(* PLC project A2ServodriveLibrary, Delta Electronics, Inc. DIADesigner-AX DIADesigner-AX 1.3, author Piotr Gliszczyński *)
(* stored: creationDateTime 2022-11-07T17:46:50.8449516, version 3.5.15.30, modificationDateTime 2022-11-07T17:45:55.5007525, organization Induprogress sp. z o.o *)
(* Library for using A2 via CiA402. For now enum for error codes processing is available. *)

{attribute 'qualified_only'}
{attribute 'strict'}
{attribute 'to_string'}
TYPE DriveA2Error : (NO_ERROR := 0, OVER_CURRENT_AL001 := 16#1, OVER_VOLTAGE_AL002 := 16#2, UNDER_VOLTAGE_AL003 := 16#3, MOTOR_COMBINATION_ERROR_AL004 := 16#4, REGENERATION_ERROR_AL005 := 16#5, OVERLOAD_AL006 := 16#6, OVERSPEED_AL007 := 16#7, ABNORMAL_PULSE_COMMAND_AL008 := 16#8, EXCESSIVE_DEVIATION_OF_POSITION_COMMAND_AL009 := 16#9, ENCODER_ERROR_AL011 := 16#11, ADJUSTMENT_ERROR_AL012 := 16#12, EMERGENCY_STOP_AL013 := 16#13, REVERSE_LIMIT_ERROR_AL014 := 16#14, FORWARD_LIMIT_ERROR_AL015 := 16#15, IGBT_OVERHEAT_AL016 := 16#16, ABNORMAL_ERROR_AL017 := 16#17, ABNORMAL_SIGNAL_OUTPUT_AL018 := 16#18, SERIAL_COMMUNICATION_ERROR_AL019 := 16#19, SERIAL_COMMUNICATION_TIME_OUT_AL020 := 16#20, MAIN_CIRCUIT_POWER_LACK_PHASE_AL022 := 16#22, EARLY_WARNING_FOR_OVERLOAD_AL023 := 16#23, ENCODER_INITIAL_MAGNETIC_FIELD_ERROR_AL024 := 16#24, THE_INTERNAL_OF_THE_ENCODER_IS_IN_ERROR_AL025 := 16#25, UNRELIABLE_INTERNAL_DATA_OF_THE_ENCODER_AL026 := 16#26, THE_INTERNAL_OF_THE_IS_IN_ERROR_AL027 := 16#27, ENCODER_VOLTAGE_ERROR_AL028 := 16#28, GRAY_CODE_ERROR_AL029 := 16#29, MOTOR_CRASH_ERROR_AL030 := 16#30, INCORRECT_WIRING_OF_THE_MOTOR_POWER_LINE_UVW_GND_AL031 := 16#31, INTERNAL_COMMUNICATION_OF_THE_ENCODER_IS_IN_ERROR_AL034 := 16#34, ENCODER_TEMPERATURE_EXCEEDS_THE_PROTECTIVE_RANGE_AL035 := 16#35, EXCESSIVE_DEVIATION_OF_FULL_CLOSED_LOOP_AL040 := 16#40, COMMUNICATION_OF_LINEAR_SCALE_IS_BREAKDOWN_AL041 := 16#41, ANALOG_INPUT_VOLTAGE_ERROR_AL042 := 16#42, WARNING_OF_SERVODRIVE_FUNCTION_OVERLOAD_AL043 := 16#43, WRONG_SETTING_OF_E_GEAR_RATIO_AL045 := 16#45, THE_ABSOLUTE_POSITION_IS_LOST_AL060 := 16#60, ENCODER_UNDER_VOLTAGE_AL061 := 16#61, THE_MULTITURN_OF_ABSOLUTE_ENCODER_OVERFLOWS_AL062 := 16#62, ENCODER_TEMPERATURE_WARNING_AL067 := 16#67, ABSOLUTE_DATA_TRANSMITTED_VIA_IO_IS_IN_ERROR_AL068 := 16#68, WRONG_MOTOR_TYPE_AL069 := 16#69, THE_ABSOLUTE_COORDINATE_HAS_NOT_BEEN_INITIALIZED_AL06A := 16#6A, ENCODER_DOES_NOT_COMPLETE_THE_COMMAND_AL070 := 16#70, ENCODER_OVERSPEED_AL072 := 16#72, ENCODER_MEMORY_ERROR_AL073 := 16#73, ABSOLUTE_ENCODER_SINGLE_TURN_POSITION_ERROR_AL074 := 16#74, ABSOLUTE_ENCODER_POSITION_ERROR_AL075 := 16#75, ENCODER_COMPUTING_ERROR_AL077 := 16#77, ENCODER_PARAMETER_ERROR_AL079 := 16#79, LOSS_OF_ENCODER_Z_PULSE_AL07A := 16#7A, ENCODER_MEMORY_BUSY_AL07B := 16#7B, COMMAND_TO_CLEAR_THE_ABSOLUTE_POSITION_ISSUED_WHEN_MOTOR_SPEED_OVER_200_RPM_AL07C := 16#7C, SERVODRIVE_POWER_IS_CYCLED_BEFORE_AL07C_IS_CLEARED_AL07D := 16#7D, ENCODER_CLEARING_PROCEDURE_ERROR_AL07E := 16#7E, SERVO_DRIVE_OUTPUTS_EXCESSIVE_CURRENT_AL083 := 16#83, REGENERATION_SETTING_ERROR_AL085 := 16#85, INPUT_VOLTAGE_IS_TOO_HIGH_AL086 := 16#86, THE_SERVO_DRIVE_DOES_NOT_CONNECT_TO_EXTERNAL_REGENERATIVE_RESISTOR_AL095 := 16#95, DSP_FIRMWARE_UPGRADE_AL099 := 16#99, CANOPEN_SDO_RECIEVES_BUFFER_OVERFLOW_AL111 := 16#111, CANOPEN_PDO_RECIEVES_BUFFER_OVERFLOW_AL112 := 16#112, INDEX_ERROR_OCCURS_WHEN_ACCESING_CANOPEN_PDO_AL121 := 16#121, SUBINDEX_ERROR_OCCURS_WHEN_ACCESING_CANOPEN_PDO_AL122 := 16#122, DATA_SIZE_ERROR_OCCURS_WHEN_ACCESING_CANOPEN_PDO_AL123 := 16#123, DATA_RANGE_ERROR_OCCURS_WHEN_ACCESING_CANOPEN_PDO_AL124 := 16#124, CANOPEN_PDO_IS_READONLY_AND_WRITE_PROTECTED_AL125 := 16#125, CANOPEN_PDO_IS_NOT_ALLOWED_IN_PDO_AL126 := 16#126, CANOPEN_PDO_IS_WRITE_PROTECTED_WHEN_SERVO_ON_AL127 := 16#127, ERROR_OCCURS_WHEN_READING_CANOPEN_PDO_VIA_EEPROM_AL128 := 16#128, ERROR_OCCURS_WHEN_WRITING_CANOPEN_PDO_VIA_EEPROM_AL129 := 16#129, THE_ACCESSING_ADDRESS_OF_EEPROM_IS_OUT_OF_RANGE_WHEN_USING_CANOPEN_PDO_AL130 := 16#130, CRC_OF_EEPROM_CALCULATION_ERROR_OCCURS_WHEN_USING_CANOPEN_PDO_AL131 := 16#131, ENTER_THE_INCORRECT_PASSWORD_WHEN_USING_CANOPEN_PDO_AL132 := 16#132, HEARTBEAT_OR_NODEGUARDING_ERROR_AL170 := 16#170, CANOPEN_PDO_TIMEOUT_AL180 := 16#180, COMMUNICATION_DISCONNECTED_AL185 := 16#185, CAN_BUS_OFF_AL186 := 16#186, ERROR_OCCURS_WHEN_LOADING_CANOPEN_DATA_AL201 := 16#201, PARAMETER_GROUP_OF_PR8_IS_OUT_OF_RANGE_AL207 := 16#207, PARAMETER_NUMBER_OF_PR8_IS_OUT_OF_RANGE_AL209 := 16#209, PARAMETER_SETTING_OF_PR8_IS_WRONG_AL213 := 16#213, WRITE_PARAMETERS_READ_ONLY_AL215 := 16#215, WRITE_PARAMETERS_PARAMETERS_LOCKED_AL217 := 16#217, SETTING_OF_MONITOR_ITEM_OF_PR8_IS_OUT_OF_RANGE_AL231 := 16#231, PR_COMMAND_OVERFLOWS_AL235 := 16#235, INDEXING_COORDINATE_IS_UNDEFINED_AL237 := 16#237, PR_POSITIONING_TIMEOUT_AL245 := 16#245, THE_NUMBER_OF_PR_COMMAND_EXCEEDS_THE_LIMIT_AL249 := 16#249, FORWARD_SOFTWARE_LIMIT_AL283 := 16#283, REVERSE_SOFTWARE_LIMIT_AL285 := 16#285, FEEDBACK_POSITION_COUNTER_OVERFLOWS_AL289 := 16#289, SERVO_OFF_ERROR_AL291 := 16#291, CANOPEN_FAILS_TO_SYNCHRONIZE_AL301 := 16#301, THE_SYNCHRONIZED_SIGNAL_OF_CANOPEN_IS_SENT_TO_FAST_AL302 := 16#302, THE_SYNCHRONIZED_SIGNAL_OF_CANOPEN_IS_SENT_TOO_SLOW_AL303 := 16#303, CANOPEN_IP_COMMAND_IS_FAILED_AL304 := 16#304, SYNC_PERIOD_IS_IN_ERROR_AL305 := 16#305, EMERGENCY_STOP_DURING_DECELERATION_AL35F := 16#35F, POSITION_DEVIATION_ALARM_FOR_DO_MC_OK_AL380 := 16#380, EMERGENCY_STOP_AL3CF := 16#3CF, CANOPEN_SYNC_FAILED_SERVO_OFF_AL3E1 := 16#3E1, CANOPEN_SYNC_SIGNAL_ERROR_SERVO_OFF_AL3E2 := 16#3E2, CANOPEN_SYNC_TIME_OUT_AL3E3 := 16#3E3, CANOPEN_IP_COMMAND_FAILED_AL3E4 := 16#3E4, SYNC_PERIOD_ERROR_AL3E5 := 16#3E5, ABSOLUTE_INDEX_COORDINATE_UNDEFINED_AL3F1 := 16#3F1, INDEX_COORDINATES_ERROR_AL400 := 16#400, NMT_RESET_COMMAND_IS_RECIEVED_WHEN_SERVO_ON_AL401 := 16#401, VALUE_OF_PR_SPECIAL_FILTER_SETTING_IS_TOO_BIG_AL404 := 16#404, SAFE_TORQUE_ENABLED_AL500 := 16#500, STO_A_LOSS_AL501 := 16#501, STO_B_LOSS_AL502 := 16#502, STO_SELF_DIAGNOSTIC_ERROR_AL503 := 16#503, SYSTEM_FAILURE_AL555 := 16#555);
END_TYPE

{attribute 'qualified_only'}
{attribute 'strict'}
{attribute 'to_string'}
TYPE DriveVFDError : (NO_ERROR := 0, OVER_CURRENT_DURING_ACCELERATION_ocA := 1, OVER_CURRENT_DURING_DECELERATION_ocd := 2, OVER_CURRENT_DURING_STEADY_OPERATION_ocn := 3, GROUND_FAULT_GFF := 4, IGBT_SHORT_CIRCUIT_BETWEEN_UPPER_BRIDGE_AND_LOWER_BRIDGE_occ := 5, OVER_CURRENT_AT_STOP_ocS := 6, OVER_VOLTAGE_DURING_ACCELERATION_ovA := 7, OVER_VOLTAGE_DURING_DECELERATION_ovd := 8, OVER_VOLTAGE_AT_CONSTANT_SPEED_ovn := 9, OVER_VOLTAGE_AT_STOP_ovS := 10, LOW_VOLTAGE_DURING_ACCELERATION_LvA := 11, LOW_VOLTAGE_DURING_DECELERATION_Lvd := 12, LOW_VOLTAGE_AT_CONSTANT_SPEED_Lvn := 13, LOW_VOLTAGE_AT_STOP_LvS := 14, PHASE_LOSS_PROTECTION_OrP := 15, IGBT_OVERHEATING_oH1 := 16, INTERNAL_KEY_PARTS_OVERHEATING_oH2 := 17, IGBT_TEMPERATURE_DETECTION_FAILURE_tH1o := 18, CAPACITOR_HARDWARE_ERROR_tH2o := 19, OVER_LOAD_oL := 21, ELECTRONIC_THERMAL_RELAY_1_PROTECTION_EoL1 := 22, ELECTRONIC_THERMAL_RELAY_2_PROTECTION_EoL2 := 23, MOTOR_OVERHEATING_oH3 := 24, OVER_TORQUE_ot1 := 26, OVER_TORQUE_ot2 := 27, UNDER_CURRENT_uC := 28, LIMIT_ERROR_LiT := 29, EEPROM_WRITE_ERROR_cF1 := 30, EEPROM_READ_ERROR_cF2 := 31, U_PHASE_ERROR_cd1 := 33, V_PHASE_ERROR_cd2 := 34, W_PHASE_ERROR_cd3 := 35, cc_HARDWARE_FAILURE_Hd0 := 36, oc_HARDWARE_ERROR_Hd1 := 37, ov_HARDWARE_ERROR_Hd2 := 38, occ_HARDWARE_ERROR_Hd3 := 39, AUTO_TUNING_ERROR_AUE := 40, PID_LOSS_ACI_AFE := 41, PG_FEEDBACK_ERROR_PGF1 := 42, PG_FEEDBACK_LOSS_PGF2 := 43, PG_FEEDBACK_STALL_PGF3 := 44, PG_SLIP_ERROR_PGF4 := 45, ACI_LOSS_ACE := 48, EXTERNAL_FAULT_EF := 49, EMERGENCY_STOP_EF1 := 50, EXTERNAL_BASE_BLOCK_bb := 51, PASSWORD_IS_LOCKED_Pcod := 52, SW_CODE_ERROR_ccod := 53, ILLEGAL_COMMAND_CE1 := 54, ILLEGAL_DATA_ADRESS_CE2 := 55, ILLEGAL_DATA_VALUE_CE3 := 56, DATA_IS_WRITTEN_TO_READ_ONLY_ADRESS_CE4 := 57, MODBUS_TRANSMISSION_TIMEOUT_CE10 := 58, BRAKE_TRANSISTOR_ERROR_bF := 60, Y_D_CONNECTION_SWITCH_ERROR_ydc := 61, DECELERATION_ENERGY_BACKUP_ERROR_dEb := 62, OVER_SLIP_ERROR_oSL := 63, ELECTRIC_VALVE_SWITCH_ERROR_ryF := 64, HARDWARE_ERROR_OF_PG_CARD_PGF5 := 65, REVERSE_DIRECTION_OF_THE_SPEED_FEEDBACK_SdRv := 68, OVER_SPEED_ROTATION_FEEDBACK_SdOr := 69, LARGE_DEVIATION_OF_SPEED_FEEDBACK_SdDe := 70, WATCHDOG_WDTT := 71, STO_LOSS_1_STL1 := 72, EMERGENCY_STOP_FOR_EXTERNAL_SAFETY_S1 := 73, EXTERNAL_BRAKE_ERROR_Brk := 75, STO_STO := 76, STO_LOSS_2_STL2 := 77, STO_LOSS_3_STL3 := 78, U_PHASE_OVER_CURRENT_BEFORE_RUN_Aoc := 79, V_PHASE_OVER_CURRENT_BEFORE_RUN_boc := 80, W_PHASE_OVER_CURRENT_BEFORE_RUN_coc := 81, OUTPUT_PHASE_LOSS_U_PHASE_OPHL := 82, OUTPUT_PHASE_LOSS_V_PHASE_OPHL := 83, OUTPUT_PHASE_LOSS_W_PHASE_OPHL := 84, PG_ABZ_LINE_OFF_AboF := 85, PG_UVW_LINE_OFF_UvoF := 86, OVERLOAD_PROTECTION_AT_LOW_FREQUENCY_oL3 := 87, ROTOR_POSITION_DETECTION_ERROR_RoPd := 89, FORCE_TO_STOP_FStp := 90, PULSE_TUNING_INDUCTANCE_L_ERROR_LEr := 92, CPU_ERROR_0_TRAP := 93, CANOPEN_GUARDING_ERROR_CGdE := 101, CANOPEN_HEARTBEAT_ERROR_CHbE := 102, CANOPEN_BUS_OFF_ERROR_CbFE := 104, CANOPEN_INDEX_ERROR_CidE := 105, CANOPEN_STATION_ADRESS_ERROR_CAdE := 106, CANOPEN_MEMORY_ERROR_CFrE := 107, INRCOM_TIMEOUT_ERROR_ictE := 111, PMLESS_SHAFT_LOCK_SfLK := 112, INTERNAL_COMMUNICATION_ERROR_CP20 := 121, INTERNAL_COMMUNICATION_ERROR_CP22 := 123, INTERNAL_COMMUNICATION_ERROR_CP30 := 124, INTERNAL_COMMUNICATION_ERROR_CP32 := 126, INTERNAL_COMMUNICATION_ERROR_CP33 := 127, OVER_TORQUE_3_ot3 := 128, OVER_TORQUE_4_ot4 := 129, INTERNAL_COMMUNICATION_ERROR_EoL3 := 134, INTERNAL_COMMUNICATION_ERROR_EoL4 := 135, oc_HARDWARE_ERROR_Hd6 := 140, GFF_OCCURS_BEFORE_RUN_b4GFF := 141, AUTOTUNE_ERROR_1_AUE1 := 142, AUTOTUNE_ERROR_2_AUE2 := 143, AUTOTUNE_ERROR_3_AUE3 := 144, AUTOTUNE_ERROR_4_AUE4 := 148, TOTAL_RESISTANCE_MEASUREMENT_FAULT_AUE5 := 149, NO_LOAD_CURRENT_IO_MEASUREMENT_FAULT_AUE6 := 150, dq_AXIS_INDUCTANCE_MEASUREMENT_FAULT_AUE7 := 151, HIGH_FREQUENCY_INJECTION_MEASUREMENT_FAULT_AUE8 := 152, PUMP_PID_FEEDBACK_ERROR_dEv := 157, CB_MISMATCH_CBM := 170, OVERPOSITION_ERROR_LIMIT_oPEE := 171);
END_TYPE

{attribute 'qualified_only'}
{attribute 'strict'}
TYPE DriveVFDWarning : (NO_WARNING := 0, COMMUNICATION_ERROR_1_CE1 := 1, COMMUNICATION_ERROR_2_CE2 := 2, COMMUNICATION_ERROR_3_CE3 := 3, COMMUNICATION_ERROR_4_CE4 := 4, COMMUNICATION_ERROR_10_CE10 := 5, SAVE_ERROR_1_SE1 := 7, SAVE_ERROR_2_SE2 := 8, IGBT_OVERHEATING_WARNING_oH1 := 9, CAPACITOR_OVERHEAT_WARNING_oH2 := 10, PID_FEEDBACK_ERROR_PID := 11, ACI_ANALOG_SIGNAL_LOSS_AnL := 12, UNDER_CURRENT_uC := 13, PG_FEEDBACK_WARNING_PGFb := 15, OVER_SPEED_WARNING_oSPd := 17, DEVIATION_WARNING_dAvE := 18, PHASE_LOSS_PHL := 19, OVER_TORQUE_1_ot1 := 20, OVER_TORQUE_2_ot2 := 21, MOTOR_OVERHEATING_oH3 := 22, OVER_SLIP_ERROR_oSL := 24, AUTO_TUNING_tUn := 25, OUTPUT_PHASE_LOSS_OPHL := 28, COPY_MODEL_ERROR_3_SE3 := 30, OVER_TORQUE_ot3 := 31, OVER_TORQUE_ot4 := 32, CANOPEN_GUARDING_TIMEOUT_CGdn := 36, CANOPEN_HEARTBEAT_ERROR_CHbn := 37, CANOPEN_BUS_OFF_ERROR_CbFn := 39, CANOPEN_INDEX_ERROR_Cldn := 40, CANOPEN_STATION_ADRESS_ERROR_CAdn := 41, CANOPEN_MEMORY_ERROR_CFrn := 42, CANOPEN_SDO_TIMEOUT_CSdn := 43, CANOPEN_SDO_RECIEVES_REGISTER_OVERFLOW_CSbn := 44, CANOPEN_STARTUP_ERROR_WARNING_Cbtn := 45, CANOPEN_FORMAT_ERROR_CPtn := 46, RTC_ADJUST_PLrA := 47, INTERCOM_ERROR_PLiC := 48, KEYPAD_RTC_TIMEOUT := 49, PLC_OPPOSITE_DEFECT_PLod := 50, PLC_SAVE_MEMORY_ERROR_PLSv := 51, DATA_DEFECT_PLdA := 52, FUNCTION_DEFECT_PLFn := 53, PLC_BUFFER_OVERFLOW_PLor := 54, FUNCTION_DEFECT_PLFF := 55, CHECKSUM_ERROR_PLSn := 56, NO_END_COMMAND_PLEd := 57, PLC_MCR_ERROR_PLCr := 58, PLCS_DOWNLOAD_FAIL_PLdF := 59, PLC_SCAN_TIME_FAIL_PLSF := 60, CAN_M_GUARDING_ERROR_PCGd := 61, CAN_M_BUS_OFF_PCbF := 62, CAN_M_NODE_LACK_PCnL := 63, CAN_M_CYCLE_TIMEOUT_PCCt := 64, CAN_M_SDO_OVER_PCSF := 65, CAN_M_SDO_TIMEOUT_PCSd := 66, CAN_M_ADRESS_ERROR_PCAd := 67, CAN_M_TIMEOUT_PCTo := 68, EXCOM_ID_FAIL_ECid := 70, EXCOM_POWER_LOSS_EXLv := 71, EXCOM_TEST_ECtt := 72, EXCOM_BUS_OFF_ECbF := 73, EXCOM_NO_POWER_ECnP := 74, EXCOM_FACTORY_DEFECT_ECFF := 75, EXCOM_INNER_ERROR_ECiF := 76, EXCOM_IO_NET_BREAK_ECio := 77, EXCOM_PARAMETER_DATA_ERROR_ECPP := 78, EXCOM_CONFIGURATION_DATA_ERROR_ECPi := 79, ETHERNET_LINK_FAIL_ECEF := 80, COMMUNICATION_TIME_OUT_ECto := 81, CHECKSUM_ERROR_ECCS := 82, RETURN_DEFECT_ECrF := 83, MODBUS_TCP_OVER_Eco0 := 84, ETHERNET_IP_OVER_ECo1 := 85, IP_FAIL_ECiP := 86, MAIL_FAIL_EC3F := 87, EXCOM_BUSY_ECbY := 88, EXCOM_CARD_BREAK_ECCb := 89, COPY_PLC_PASSWORD_ERROR_CPLP := 90, COPY_PLC_READ_MODE_ERROR_CPL0 := 91, COPY_PLC_WRITE_MODE_CPL1 := 92, COPY_CPL_VERSION_ERROR_CPLv := 93, COPY_PLC_SIZE_ERROR_CPLS := 94, COPY_PLC_PLC_FUNCTION_CPLF := 95, COPY_PLC_TIMEOUT_CPLt := 96, INCROM_TIMEOUT_ictn := 101, DECELERATION_ENERGY_BACKUP_ERROR_dEb := 102, PID_FEEDBACK_FAULT_dEv := 103, EXTIMATED_SPEED_REVERSE_SpdR := 105, DECELERATION_ENERGY_BACKUP_dEb := 123, INDEX_PULSE_FAIL_INDX := 125, NOT_HOME_YET_nHoY := 126, HW_POS_LIMIT_HPL := 127, HW_NEG_LIMIT_HnL := 128, SW_POS_LIMIT_SPL := 129, SW_NEG_LIMIT_SnL := 130, POSN_OVERFLOW_PoF := 131, HOME_PROC_FAULT_HPF := 132, OVER_POS_ERR_LIM_Ope := 133);
END_TYPE
